FUNCTION_BLOCK SS3_ifb_flipper (* Basic FB with empty ECC *)
  (* Standard: 61499-2 *)
  (* Version 1.0, 2025-05-16, DEVIASH *)
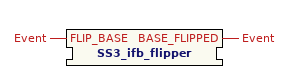
  EVENT_INPUT
    FLIP_BASE;
  END_EVENT
  EVENT_OUTPUT
    BASE_FLIPPED;
  END_EVENT
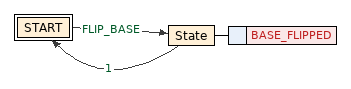
  EC_STATES
    START; (* Initial State *)
    State : -> BASE_FLIPPED;
  END_STATES
  EC_TRANSITIONS
    START TO State := FLIP_BASE;
    State TO START := 1;
  END_TRANSITIONS
END_FUNCTION_BLOCK
